(* IEC 61131-3 sources: Word/plc-course/06-edges-and-one-shots/labs/starter, 3 files *)

(* ---- 06-1-toggle-lamp.st ---- *)
(* Lab 06-1: One-button floodlight toggle (push-on / push-off).
   Module 06 (Edge detection and one-shots). STARTER - the declarations are done
   for you; write the logic where it says TODO, then run:
     python3 tools/plctest.py 06-edges-and-one-shots/labs/starter/06-1-toggle-lamp.st *)

PROGRAM ToggleLamp
  VAR (* I/O - addresses follow the OpenPLC convention *)
    LightPB      AT %IX0.0 : BOOL;  (* Floodlight push-button, NO: TRUE while pressed *)
    LightsEnable AT %IX0.1 : BOOL;  (* Gatehouse key switch: TRUE = bay lighting enabled *)
    Floodlight   AT %QX0.0 : BOOL;  (* Floodlight contactor coil *)
  END_VAR
  VAR (* internal - add your own variables here (an R_TRIG instance, or a
         "previous value" bit) *)
    Spare : BOOL;
  END_VAR

  (* TODO: replace this placeholder with your logic.
     Each PRESS of LightPB must toggle Floodlight, however long it is held.
     LightsEnable = FALSE forces the light off and ignores the button. *)
  Floodlight := FALSE;
END_PROGRAM

CONFIGURATION Config0
  RESOURCE Res0 ON PLC
    TASK MainTask(INTERVAL := T#10ms, PRIORITY := 0);
    PROGRAM Inst0 WITH MainTask : ToggleLamp;
  END_RESOURCE
END_CONFIGURATION

(* ---- 06-2-event-counter.st ---- *)
(* Lab 06-2: Carton and product-change counter (event counting and change-of-value).
   Module 06 (Edge detection and one-shots). STARTER - the declarations are done
   for you; write the logic where it says TODO, then run:
     python3 tools/plctest.py 06-edges-and-one-shots/labs/starter/06-2-event-counter.st *)

PROGRAM EventCounter
  VAR (* I/O - addresses follow the OpenPLC convention *)
    PartPE  AT %IX0.0 : BOOL;  (* Photo-eye: TRUE while a carton blocks the beam *)
    ResetPB AT %IX0.1 : BOOL;  (* Count reset push-button, NO: TRUE while pressed *)
  END_VAR
  VAR (* HMI values - part of the lab interface *)
    ProductSel : INT;          (* Product number selected by the operator on the HMI, 1..4 *)
    PartCount  : DINT;         (* Cartons counted since the last reset *)
    SelChanges : INT;          (* Changes of ProductSel since the last reset *)
  END_VAR
  VAR (* internal - add your own variables here: edge detectors, "previous
         value" variables, a first-scan flag ... *)
    Spare : BOOL;
  END_VAR

  (* TODO: replace these placeholders with your logic.
     - PartCount: +1 for every carton that ARRIVES at the photo-eye.
     - SelChanges: +1 for every change of ProductSel.
     - The input values present at power-up are not events.
     - ResetPB: counts are 0 while it is held; nothing is counted meanwhile,
       and nothing is counted "late" when it is released. *)
  PartCount := 0;
  SelChanges := 0;
END_PROGRAM

CONFIGURATION Config0
  RESOURCE Res0 ON PLC
    TASK MainTask(INTERVAL := T#10ms, PRIORITY := 0);
    PROGRAM Inst0 WITH MainTask : EventCounter;
  END_RESOURCE
END_CONFIGURATION

(* ---- 06-3-duty-standby.st ---- *)
(* Lab 06-3: Duty-standby pump alternation.
   Module 06 (Edge detection and one-shots). STARTER - the declarations are done
   for you; write the logic where it says TODO, then run:
     python3 tools/plctest.py 06-edges-and-one-shots/labs/starter/06-3-duty-standby.st
   Training exercise only: a real pump station also needs level alarms, run
   feedback, start delays and a design review (Modules 07, 14, 16). *)

PROGRAM DutyStandby
  VAR (* I/O - addresses follow the OpenPLC convention *)
    Demand     AT %IX0.0 : BOOL;  (* Pumping demand from the sump level control: TRUE = pump needed *)
    Pump1OK_NC AT %IX0.1 : BOOL;  (* Pump 1 healthy (overload relay + motor protection), NC: TRUE when healthy *)
    Pump2OK_NC AT %IX0.2 : BOOL;  (* Pump 2 healthy, NC: TRUE when healthy *)
    Pump1      AT %QX0.0 : BOOL;  (* Pump 1 contactor *)
    Pump2      AT %QX0.1 : BOOL;  (* Pump 2 contactor *)
  END_VAR
  VAR (* internal - add your own variables here: an edge detector for the
         demand, the selected pump, which pump ran last ... *)
    Spare : BOOL;
  END_VAR

  (* TODO: replace these placeholders with your logic.
     - Each NEW demand starts the pump that did not run last time
       (Pump 1 first after power-up).
     - A faulted pump is never started; the other one runs instead.
     - Never both pumps at once. *)
  Pump1 := FALSE;
  Pump2 := FALSE;
END_PROGRAM

CONFIGURATION Config0
  RESOURCE Res0 ON PLC
    TASK MainTask(INTERVAL := T#10ms, PRIORITY := 0);
    PROGRAM Inst0 WITH MainTask : DutyStandby;
  END_RESOURCE
END_CONFIGURATION
